FUNCTION_BLOCK EcMasterFrameCount IMPLEMENTS IEcTask
VAR_INPUT
END_VAR
VAR_OUTPUT
END_VAR
VAR
	iState : INT;
	masterFrameCount : Tc2_EtherCAT.FB_EcMasterFrameCount;
	_execute: BOOL;
	_done: BOOL;
	_busy: BOOL;
	_error: BOOL;
	_netId: AMSNETID;
END_VAR

CASE iState OF
	0:
		IF _execute THEN
			_done := FALSE;
			_busy := TRUE;
			_error := FALSE;
			masterFrameCount.bExecute := TRUE;
			IF masterFrameCount.bBusy THEN
				iState := 10;
				_execute := false;
			END_IF
		END_IF
	10:
		IF NOT masterFrameCount.bBusy THEN
			IF NOT masterFrameCount.bError THEN
				_done := TRUE;
			ELSE
				_error := TRUE;
			END_IF
			_busy := FALSE;
			masterFrameCount.bExecute := FALSE;
			iState := 0;
		END_IF
END_CASE

masterFrameCount(sNetId := Tc2_System.F_CreateAmsNetId(nIds := NetId));

{warning 'add method implementation '}
METHOD Abort : BOOL
masterFrameCount.bExecute := FALSE;
_busy := FALSE;
_execute := FALSE;
Abort := TRUE;
iState := 0;
END_METHOD

{warning 'add property implementation'}
PROPERTY Busy : BOOL
GET
Busy := _busy;
END_GET
END_PROPERTY

{warning 'add property implementation'}
PROPERTY Done : BOOL
GET
Done := _done;
END_GET
END_PROPERTY

{warning 'add property implementation'}
PROPERTY Error : BOOL
GET
Error := _error;
END_GET
END_PROPERTY

{warning 'add method implementation '}
METHOD Execute : BOOL
IF NOT masterFrameCount.bBusy THEN
	Execute := _execute := True;
END_IF
END_METHOD

PROPERTY FrameNumber : UDINT
GET
FrameNumber := masterFrameCount.nFrames;
END_GET
END_PROPERTY

{warning 'add property implementation'}
PROPERTY NetID : amsnetid
GET
NetID := _netId;
END_GET
SET
_netId := NetID;
END_SET
END_PROPERTY

END_FUNCTION_BLOCK

(* stored: Version 1.1.0.1, ProductVersion 3.1.4024.11
   POU EcMasterFrameCount: Id {370d08c0-f5dd-4344-88db-4613da35681b}, SpecialFunc None
   Method Abort: Id {093c7b74-45db-4148-bc3f-149f7eefe1a9}
   Property Busy: Id {b57ab63a-5198-4ab9-a9a5-110895a21ede}
   Get Get: Id {50637dbe-9d73-44bd-a1b9-1111785940c2}
   Property Done: Id {12d7aacb-4719-4359-a3a3-6402d220140d}
   Get Get: Id {6ed416b9-8cdf-44ec-91e6-caaa4a5af74c}
   Property Error: Id {2c2312b8-9992-4728-9e8b-27705800aec8}
   Get Get: Id {1c71a323-64c1-42be-bcf4-2adc9aebf46d}
   Method Execute: Id {0a234463-2f27-4bd4-821d-d0e8716e3ce6}
   Property FrameNumber: Id {2efbfa2e-ac11-4e4e-b8d2-39a53470a14a}
   Get Get: Id {9108cf7f-ee48-4eec-abc3-9552ed79daf8}
   Property NetID: Id {740776fd-9c29-4801-baf8-74a1e95301e8}
   Get Get: Id {b538d0a1-da1c-4bd4-ad15-95be6377d3fb}
   Set Set: Id {8126ca2a-9d5e-4fc4-b8d5-c4f46adb3b07} *)
